(*
version 1.0	21 feb 2008
programmer 	hugo
tested by		oscat

this function calculates the cosinus function of a complex number

*)
FUNCTION CCOS : complex
VAR_INPUT
	X : complex;
END_VAR

CCOS := CCOSH(CSET(-X.im, X.re));


(* revision history
hm	21. feb 2008	rev 1.0
	original version

*)

END_FUNCTION

(* stored: Version 1.1.0.1
   POU CCOS: Id {a5792ea0-5fb4-46c9-8425-179d4843cb5d}, SpecialFunc None *)
